{attribute 'enable_dynamic_creation'}
FUNCTION_BLOCK Node IMPLEMENTS IListItem
VAR_IN_OUT
//	data : INT;
//	next : POINTER TO Node;
END_VAR

PROPERTY data : INT
GET
END_GET
SET
END_SET
END_PROPERTY

PROPERTY next : POINTER TO Node
GET
END_GET
SET
END_SET
END_PROPERTY

END_FUNCTION_BLOCK

(* stored: Version 1.1.0.1, ProductVersion 3.1.4024.11
   POU Node: Id {6ca422d5-da8c-4e56-80fb-ca3392e57996}, SpecialFunc None
   Property data: Id {42a49789-e337-478f-90a9-4d174f51e741}
   Get Get: Id {1cfacef1-85f0-4696-8a9c-29e617b1bdf3}
   Set Set: Id {d4edf611-b6c6-4a37-bed1-5d4e3a7397f6}
   Property next: Id {d1234b62-4117-4ed7-94bb-47bc3d3babca}
   Get Get: Id {72b192ab-da2a-439b-87f7-53e0adca7535}
   Set Set: Id {2452b0f3-a460-4a29-90a9-b627107e255e} *)
